(* CoDeSys 2.3 export: E_SENSOR.EXP *)

(* Data type *)
TYPE E_Sensor : (
	Thermokon_MDS := 1,
	Thermokon_FTW04VV := 2,
	PT1000 := 3
);
END_TYPE
